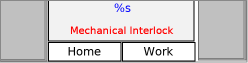
VISUALIZATION Std_Cylinder_Ctrl  // 248x63
VAR_IN_OUT
	m_Input_Inst : None;
END_VAR
    RoundedRectangle (48,0 146x41), "%s", text variable: m_Input_Inst.IN_CylName
    RoundedRectangle (48,42 73x19), "Home", colour toggle: (m_Input_Inst.S_HomePos) <> 0, invisible if: (m_Input_Inst.E_HomeErr) <> 0
    RoundedRectangle (122,42 73x19), "Work", colour toggle: (m_Input_Inst.S_WorkPos) <> 0, invisible if: (m_Input_Inst.E_WorkErr) <> 0
    Group (-1,0 46x59)
        tap m_Input_Inst.T_ManHome
        Button (0,0 48x61)
            tap m_Input_Inst.In_ManHome
        Polygon (38,51)
        Polygon (35,51)
    Group (198,0 46x59)
        tap m_Input_Inst.T_ManWork
        Button (0,0 48x60)
            tap m_Input_Inst.In_ManWork
        Polygon (10,50)
        Polygon (13,50)
    RoundedRectangle (49,21 146x19), "Mechanical Interlock", invisible if: (NOT (NOT m_Input_Inst.In_WorkXLock AND m_Input_Inst.T_ManWork)) <> 0
    RoundedRectangle (49,21 146x19), "Mechanical Interlock", invisible if: (NOT (NOT m_Input_Inst.In_HomeXLock AND m_Input_Inst.T_ManHome)) <> 0
    RoundedRectangle (48,42 73x19), "Home", colour toggle: (m_Input_Inst.E_HomeErr) <> 0, invisible if: (NOT m_Input_Inst.E_HomeErr) <> 0
    RoundedRectangle (122,42 73x19), "Work", colour toggle: (m_Input_Inst.E_WorkErr) <> 0, invisible if: (NOT m_Input_Inst.E_WorkErr) <> 0
END_VISUALIZATION

(* stored: Version 1.1.0.1, ProductVersion 3.1.4018.2
   Visu Std_Cylinder_Ctrl: Id {004f8440-9982-4ee8-bc5f-430e8b6cc30d} *)
